SUBAPPLICATION Uebung_001 (* Subapplication Type *)
  (* Standard: 61499-2 *)
  (* Version 1.0, 2023-10-23, franz *)
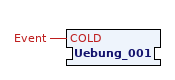
  EVENT_INPUT
    COLD;
  END_EVENT
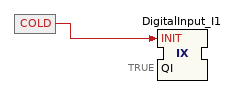
  FBS
    DigitalInput_I1 : IX(QI := TRUE);
  END_FBS
  EVENT_CONNECTIONS
    COLD TO DigitalInput_I1.INIT;
  END_CONNECTIONS
END_SUBAPPLICATION
